PROGRAM Main
VAR
	{attribute 'pytmc' := '
        pv: TST:PPM:MMS:01
		io: io
	'}
	{attribute 'TcLinkTo' := '.bLimitForwardEnable  := TIIB[EL7041]^STM Status^Status^Digital input 1;
	                          .bLimitBackwardEnable := TIIB[EL7041]^STM Status^Status^Digital input 2;
	                          .bBrakeRelease        := TIIB[EL2004]^Channel 1^Output'}
	M1: DUT_MotionStage;
	
	{attribute 'pytmc' := '
		pv: TST:PPM
		io: io
	'}
	{attribute 'TcLinkTo' := '.fbGige.iIlluminatorINT := TIIB[EL4004]^AO Outputs Channel 1^Analog output;
	                          .fbGige.bGigePower := TIIB[EL2004]^Channel 2^Output;
							  .fbPowerMeter.iVoltageINT := TIIB[EL3062]^AI Standard Channel 1^Value;
							  .fbPowerMeter.fbThermoCouple.bError := TIIB[EL3314]^TC Inputs Channel 1^Status^Error;
							  .fbPowerMeter.fbThermoCouple.bUnderrange := TIIB[EL3314]^TC Inputs Channel 1^Status^Underrange;
							  .fbPowerMeter.fbThermoCouple.bOverrange := TIIB[EL3314]^TC Inputs Channel 1^Status^Overrange;
							  .fbPowerMeter.fbThermoCouple.iRaw := TIIB[EL3314]^TC Inputs Channel 1^Value;
							  .fbYagThermoCouple.bError := TIIB[EL3314]^TC Inputs Channel 2^Status^Error;
							  .fbYagThermoCouple.bUnderrange := TIIB[EL3314]^TC Inputs Channel 2^Status^Underrange;
							  .fbYagThermoCouple.bOverrange := TIIB[EL3314]^TC Inputs Channel 2^Status^Overrange;
							  .fbYagThermoCouple.iRaw := TIIB[EL3314]^TC Inputs Channel 2^Value'}
	fbPPM: FB_PPM;
	
	{attribute 'pytmc' := '
		pv: TST:PPM:MMS:01:ENC_RAW
		io: i
	'}
	iAdjustedEncoder: UDINT;
	iRawEncoder AT %I*: ULINT;
	iMaxLINT: ULINT := 18446744073709551615;
END_VAR

fbPPM(stYStage := M1);
M1.bHardwareEnable := TRUE;
iAdjustedEncoder :=  ULINT_TO_UDINT(iMaxLINT - iRawEncoder);

END_PROGRAM

(* stored: Version 1.1.0.1, ProductVersion 3.1.4022.12
   POU Main: Id {cb921465-efa3-4bda-880b-e8f57acf61aa}, SpecialFunc None *)
